Staubli VAL3: start.pgx

program start()
  local num l_nLastId
  local num l_ni
begin
  call Init()
  taskCreate "light",30,ContorlLight()
  wait(taskStatus("light")==1)
  call Main()
end
